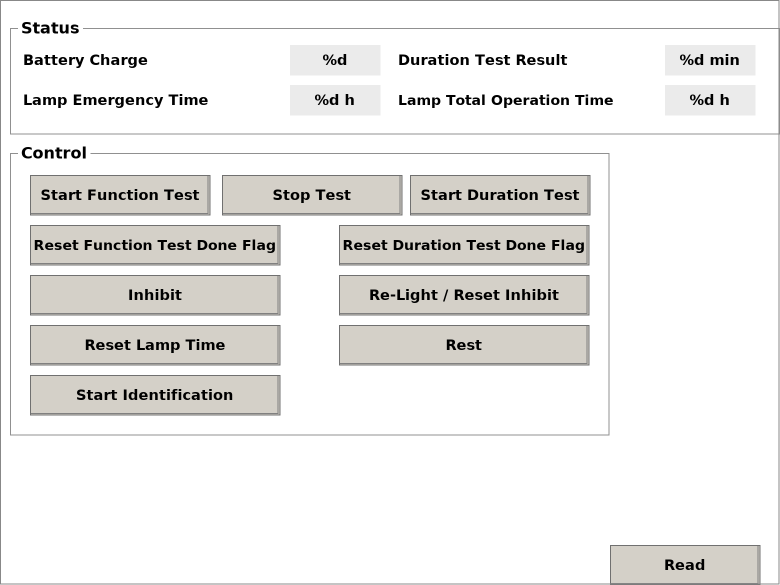
VISUALIZATION Visu_Part202Commands  // 780x585
    GroupBox (10,145 599x290), "Control"
        Button (20,130 250x40), "Inhibit"
            OnMouseClick: execute { DALI_Commissioning.fbPart202Emergency.bInhibit := TRUE; }
        Button (20,80 250x40), "Reset Function Test Done Flag"
            OnMouseClick: execute { DALI_Commissioning.fbPart202Emergency.bResetFunctionTestDoneFlag := TRUE; }
        Button (20,30 180x40), "Start Function Test"
            OnMouseClick: execute { DALI_Commissioning.fbPart202Emergency.bStartFunctionTest := true; }
        Button (20,180 250x40), "Reset Lamp Time"
            OnMouseClick: execute { DALI_Commissioning.fbPart202Emergency.bResetLampTime := TRUE; }
        Button (20,230 250x40), "Start Identification"
            OnMouseClick: execute { DALI_Commissioning.fbPart202Emergency.bStartIdentification := TRUE; }
        Button (212,30 180x40), "Stop Test"
            OnMouseClick: execute { DALI_Commissioning.fbPart202Emergency.bStopTest := TRUE; }
        Button (400,30 180x40), "Start Duration Test"
            OnMouseClick: execute { DALI_Commissioning.fbPart202Emergency.bStartDurationTest := TRUE; }
        Button (329,130 250x40), "Re-Light / Reset Inhibit"
            OnMouseClick: execute { DALI_Commissioning.fbPart202Emergency.bResetInhibit := TRUE; }
    GroupBox (10,20 770x114), "Status"
        Textfield (385,65 220x30), "Lamp Total Operation Time"
        Textfield (655,65 90x30), "%d h", text variable: DALI_Commissioning.fbPart202Emergency.nLampTotalOperationTime
        Textfield (655,25 90x30), "%d min", text variable: DALI_Commissioning.fbPart202Emergency.nDurationTestResult
        Textfield (280,65 90x30), "%d h", text variable: DALI_Commissioning.fbPart202Emergency.nLampEmergencyTime
        Textfield (280,25 90x30), "%d", text variable: DALI_Commissioning.fbPart202Emergency.nBatteryCharge
        Textfield (10,25 220x30), "Battery Charge"
        Textfield (10,65 220x30), "Lamp Emergency Time"
        Textfield (385,25 220x30), "Duration Test Result"
    Button (339,225 250x40), "Reset Duration Test Done Flag"
        OnMouseClick: execute { DALI_Commissioning.fbPart202Emergency.bResetDurationTestDoneFlag := TRUE; }
    Button (339,325 250x40), "Rest"
        OnMouseClick: execute { DALI_Commissioning.fbPart202Emergency.bRest := TRUE; }
    Button (610,545 150x40), "Read"
        OnMouseClick: execute { DALI_Commissioning.fbPart202Emergency.bReadCommands:=TRUE; }
END_VISUALIZATION

(* stored: Version 1.1.0.1, ProductVersion 3.1.4024.12
   Visu Visu_Part202Commands: Id {85589b74-1813-4046-a0a0-755120ce2310} *)
